FUNCTION Convert_UDINT_TO_USINT : Hresult
VAR_INPUT
	in : UDINT;
	out : REFERENCE TO USINT;
END_VAR
VAR
	converted : USINT;
END_VAR
VAR CONSTANT
	INCOMPATIBLE : HRESULT := 16#9811070E;
END_VAR

converted := UDINT_TO_USINT(in);

IF (USINT_TO_UDINT(converted) <> in) THEN
	Convert_UDINT_TO_USINT := INCOMPATIBLE;
	RETURN;
END_IF

out := converted;

END_FUNCTION

(* stored: Version 1.1.0.1, ProductVersion 3.1.4024.12
   POU Convert_UDINT_TO_USINT: Id {69d13335-da94-4aa7-92da-1c956adb95b8}, SpecialFunc None *)
